Staubli VAL3: read_ID.pgx

public program read_ID()
  local bool non_stop
begin

  non_stop = true

  do

    putln(getMoveId())
    putln(getMonitorSpeed())

  until non_stop != true

end
